// TIA Portal V16 export
// export: Created 2021-09-08T12:46:12.2706285Z, ExportSetting WithDefaults, DisplayName Totally Integrated Automation Portal, DisplayVersion V16 Update 3, DisplayName TIA Portal Version Control Interface, DisplayVersion V16 Update 2, DisplayName TIA Portal Openness, DisplayVersion V16 Update 3, DisplayName TIA Portal Teamcenter Gateway, DisplayVersion V16, DisplayName STEP 7 Professional, DisplayVersion V16 Update 3, DisplayName STEP 7 Safety, DisplayVersion V16, DisplayName WinCC Advanced, DisplayVersion V16 Update 3
FUNCTION_BLOCK "DigitalSensorCntrl"   // FB80, FBD
{ S7_Optimized_Access := 'TRUE' }
VERSION : 0.1
// выход 1-авария
// в режиме авто, прямой вход - 0-авария, с инверсией - 1-авария
// в ручном режиме включение авария -
// stored: AutoNumber false, IsIECCheckEnabled false, IsRetainMemResEnabled false, MemoryReserve 100, SetENOAutomatically false, UDAEnableTagReadback false
   VAR_INPUT
      i : Bool;
   END_VAR
   VAR_IN_OUT
      sensor : "digitalSensor";
   END_VAR
BEGIN

REGION Network 1: Промежуточное состояние без задержки
   // 1-alarm
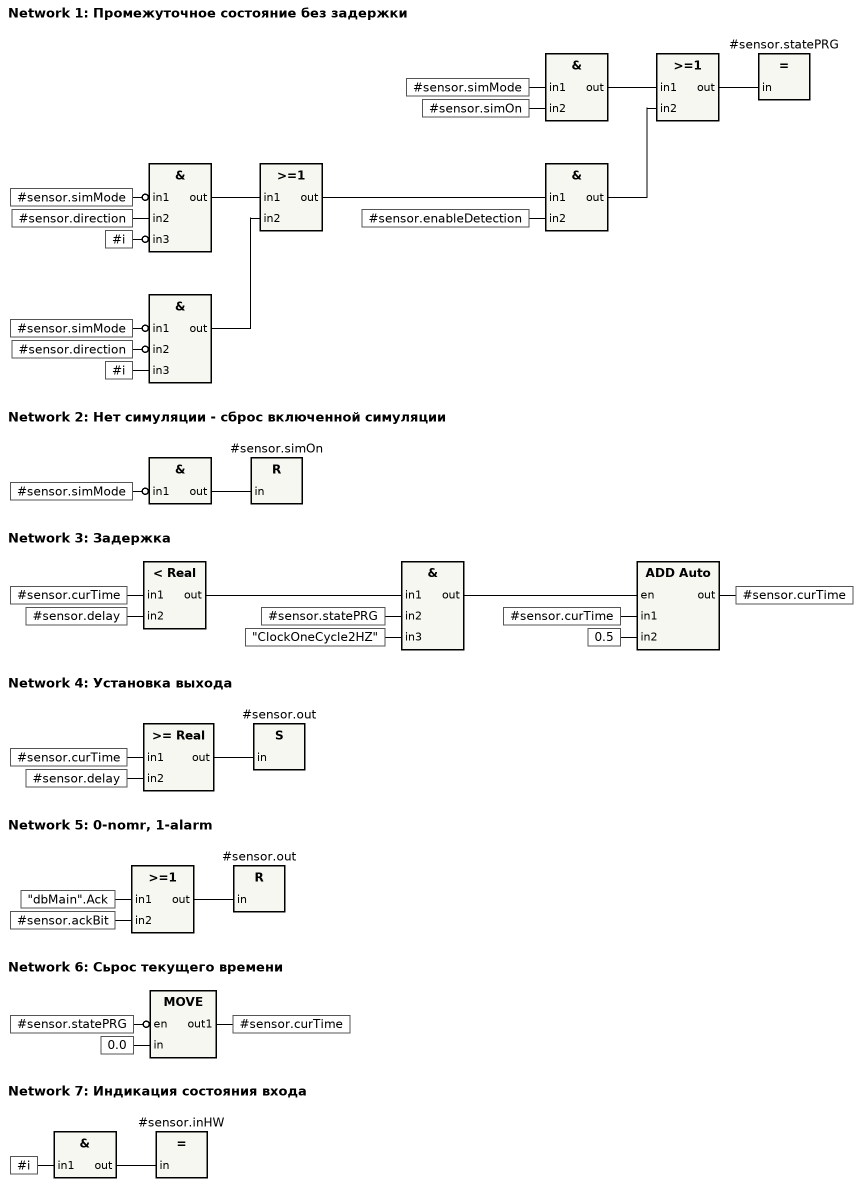
   #sensor.statePRG := (#sensor.simMode AND #sensor.simOn) OR (((NOT #sensor.simMode AND #sensor.direction AND NOT #i) OR (NOT #sensor.simMode AND NOT #sensor.direction AND #i)) AND #sensor.enableDetection);
END_REGION

REGION Network 2: Нет симуляции - сброс включенной симуляции
   IF NOT #sensor.simMode THEN #sensor.simOn := FALSE; END_IF;
END_REGION

REGION Network 3: Задержка
   IF (#sensor.curTime < #sensor.delay) AND #sensor.statePRG AND "ClockOneCycle2HZ" THEN
       #sensor.curTime := #sensor.curTime + 0.5;
   END_IF;
END_REGION

REGION Network 4: Установка выхода
   IF #sensor.curTime >= #sensor.delay THEN #sensor.out := TRUE; END_IF;
END_REGION

REGION Network 5: 0-nomr, 1-alarm
   IF "dbMain".Ack OR #sensor.ackBit THEN #sensor.out := FALSE; END_IF;
END_REGION

REGION Network 6: Сьрос текущего времени
   IF NOT #sensor.statePRG THEN #sensor.curTime := 0.0; END_IF;
END_REGION

REGION Network 7: Индикация состояния входа
   #sensor.inHW := #i;
END_REGION
END_FUNCTION_BLOCK
